{attribute 'qualified_only'}
{attribute 'strict'}
TYPE eIoTCommVersion :
(
	V1 := 0,
	V2 := 1
);
END_TYPE

(* stored: Version 1.1.0.1, ProductVersion 3.1.4026.18
   DUT eIoTCommVersion: Id {f890216b-e8c2-4bcb-8a19-1ba9157488c4} *)
